FUNCTION_BLOCK FB_PLCTime
VAR_INPUT
END_VAR
VAR_OUTPUT
	sTime				: STRING;
END_VAR
VAR
	fbGetTime			: NT_GetTime;
	TimeStr				: TIMESTRUCT;
END_VAR

fbGetTime(
	START := TRUE,
	NETID := '',
	TIMESTR => TimeStr
	);
fbGetTime(
	START := FALSE,
	NETID := ''
	);
	
sTime := CONCAT(TO_STRING(TimeStr.wHour), ':'); 
IF TimeStr.wMinute < 10 THEN
	sTime := CONCAT(sTime, '0');
	sTime := CONCAT(sTime, TO_STRING(TimeStr.wMinute));
ELSE
	sTime := CONCAT(sTime, TO_STRING(TimeStr.wMinute));	
END_IF 
sTime := CONCAT(sTime, ':');
IF TimeStr.wSecond < 10 THEN
	sTime := CONCAT(sTime, '0');
	sTime := CONCAT(sTime, TO_STRING(TimeStr.wSecond));
ELSE
	sTime := CONCAT(sTime, TO_STRING(TimeStr.wSecond));	
END_IF
sTime := CONCAT(sTime, '.');
sTime := CONCAT(sTime, TO_STRING(TimeStr.wMilliseconds));

END_FUNCTION_BLOCK

(* stored: Version 1.1.0.1, ProductVersion 3.1.4024.2
   POU FB_PLCTime: Id {a5d7e61a-069c-4933-9ab6-1c2c5894ac9a}, SpecialFunc None *)
